FUNCTION_BLOCK EcMasterGetDeviceId IMPLEMENTS IEcTask
VAR_INPUT
END_VAR
VAR_OUTPUT
END_VAR
VAR
	iState : INT;
	getDeviceIdentity : Tc2_EtherCAT.FB_EcGetSlaveIdentity;
	_execute: BOOL;
	_done: BOOL;
	_busy: BOOL;
	_error: BOOL;
	_netId: AMSNETID;
END_VAR

CASE iState OF
	0:
		IF _execute THEN
			_done := FALSE;
			_busy := TRUE;
			_error := FALSE;
			getDeviceIdentity.bExecute := TRUE;
			IF getDeviceIdentity.bBusy THEN
				iState := 10;
				_execute := false;
			END_IF
		END_IF
	10:
		IF NOT getDeviceIdentity.bBusy THEN
			IF NOT getDeviceIdentity.bError THEN
				_done := TRUE;
			ELSE
				_error := TRUE;
			END_IF
			_busy := FALSE;
			getDeviceIdentity.bExecute := FALSE;
			iState := 0;
		END_IF
END_CASE

getDeviceIdentity(sNetId := Tc2_System.F_CreateAmsNetId(nIds := NetId));

{warning 'add method implementation '}
METHOD Abort : BOOL
getDeviceIdentity.bExecute := FALSE;
_busy := FALSE;
_execute := FALSE;
Abort := TRUE;
iState := 0;
END_METHOD

{warning 'add property implementation'}
PROPERTY Busy : BOOL
GET
Busy := _busy;
END_GET
END_PROPERTY

PROPERTY DeviceAddr : uint
GET
DeviceAddr := getDeviceIdentity.nSlaveAddr;
END_GET
SET
getDeviceIdentity.nSlaveAddr := DeviceAddr;
END_SET
END_PROPERTY

PROPERTY DeviceIdentity : ST_EcSlaveIdentity
GET
DeviceIdentity := getDeviceIdentity.identity;
END_GET
END_PROPERTY

{warning 'add property implementation'}
PROPERTY Done : BOOL
GET
Done := _done;
END_GET
END_PROPERTY

{warning 'add property implementation'}
PROPERTY Error : BOOL
GET
Error := _error;
END_GET
END_PROPERTY

{warning 'add method implementation '}
METHOD Execute : BOOL
IF NOT getDeviceIdentity.bBusy THEN
	Execute := _execute := true;
END_IF
END_METHOD

{warning 'add property implementation'}
PROPERTY NetID : amsnetid
GET
NetID := _netId;
END_GET
SET
_netId := NetID;
END_SET
END_PROPERTY

END_FUNCTION_BLOCK

(* stored: Version 1.1.0.1, ProductVersion 3.1.4024.9
   POU EcMasterGetDeviceId: Id {da1da148-5d06-44ce-88ec-731d976d6b8d}, SpecialFunc None
   Method Abort: Id {af12244c-3ccd-4164-b8b6-c4c53fe0cb02}
   Property Busy: Id {1858ae8f-d8a9-4f20-98f2-e8b1f464c234}
   Get Get: Id {25c198a7-7a2b-4e21-b4d4-906f3c677d67}
   Property DeviceAddr: Id {3ee2e69f-a4a0-48ce-971a-1961ee85cc68}
   Get Get: Id {4acea6b1-ab62-4ab7-a72f-56db9a45e7e8}
   Set Set: Id {4a37f428-76b4-407b-925d-4646493d8d5e}
   Property DeviceIdentity: Id {e32086c0-3244-4aae-9191-a84993f75800}
   Get Get: Id {7e613b50-9b5b-4549-afed-76d6ed5f72df}
   Property Done: Id {83aadf5b-d4ca-439d-b818-777c7807bc5e}
   Get Get: Id {22fad5ad-2404-4570-9671-83645f3a3b9b}
   Property Error: Id {11c09dfd-370c-4119-a58f-3e3bdf01bdd4}
   Get Get: Id {769b4165-d3af-4e0e-9fa2-dc7390d73bc4}
   Method Execute: Id {87b62678-26b8-41f6-aec2-2a5e192c4360}
   Property NetID: Id {0363d4d3-a94a-40e3-b3ff-8cf0804bf878}
   Get Get: Id {376ad78c-fce0-4480-b230-839aec19637d}
   Set Set: Id {a92c6f9f-d6c0-49b2-88b0-7da6b25ac1e0} *)
